(* CODESYS project RobotArm.project

Project tree, tasks and I/O mapping:
  Device : CODESYS Control for Raspberry Pi SL, 3S - Smart Software Solutions GmbH, version 3.5.12.0
    application Application
      libraries: Standard, * (System); SysProcess, 3.5.7.0 (System); SysTypes Interfaces, 3.5.2.0 (System)
      task MainTask (cyclic, interval t#10ms, priority 1) calls PLC_PRG
      task VISU_TASK (cyclic, interval 100 ms, priority 31) calls VisuElems.Visu_Prg
      program PLC_PRG [ST]
      program prgModeSelect [ST]
      program prgStartup [CFC]
      visualisation Visualization
      GVLs/
        global variables GVL_IO
        global variables GVL_Constants
        global variables GVL_Axis
      DUTs/
        data type eAxis
      FBs/
        function block fb_AxisControl [CFC]
        function block fb_FreeMode [SFC]: MoveA_active, MoveA_exit, Check_active
      program prgAxisControl [ST]
    SoftMotion General Axis Pool
    I²C
      I2C_master : I2C master, 3S - Smart Software Solutions GmbH, version 1.0.0.0
        Adafruit_PWM_SoftMotion : Adafruit PWM SoftMotion, 3S - Smart Software Solutions GmbH, version 1.2.0.0
            settings: I²C address = 16#40; Frequency [Hz] = 60
          SM_Drive_Servo_Base : SM_Drive_Servo, 3S - Smart Software Solutions GmbH, version 3.5.11.0
              settings: wDriveID = 0; fSWMaxVelocity = 1000; Commisioning.smci.Distance = 10; Commisioning.smci.Velocity = 30; Commisioning.smci.Acceleration = 500; Commisioning.smci.Deceleration = 500; negative position [units] = -90; positive position [units] = 100; minimum signal length [ms] = 0.5; maximum signal length [ms] representing the positive position = 2.2
          SM_Drive_Servo_Upright : SM_Drive_Servo, 3S - Smart Software Solutions GmbH, version 3.5.11.0
              settings: fSWMaxVelocity = 1000; negative position [units] = -90; positive position [units] = 100; minimum signal length [ms] = 0.5; maximum signal length [ms] representing the positive position = 2.2
          SM_Drive_Servo_Arm : SM_Drive_Servo, 3S - Smart Software Solutions GmbH, version 3.5.11.0
              settings: wDriveID = 2; fSWMaxVelocity = 1000
          SM_Drive_Servo_Gripper : SM_Drive_Servo, 3S - Smart Software Solutions GmbH, version 3.5.11.0
              settings: wDriveID = 3; fSWMaxVelocity = 1000
    SPI
    GPIOs_A_B : GPIOs B+/Pi2, 3S - Smart Software Solutions GmbH, version 3.5.11.0
        unmapped channels: digital inputs (GPIO0..GPIO31), digital outputs (GPIO0..GPIO31)
    Onewire
    Camera device
      <Empty>
  text list GlobalTextList
*)

// Device/Application/DUTs/eAxis
TYPE eAxis :
(
	Base := 1,
	Upright := 2,
	Arm := 3,
	Gripper := 4
);
END_TYPE

// Device/Application/GVLs/GVL_IO
VAR_GLOBAL
	rVelocity : LREAL := 100;
	rPos : ARRAY [1..iNoOfAxis] OF LREAL;
END_VAR

// Device/Application/GVLs/GVL_Constants
VAR_GLOBAL CONSTANT
	iNoOfAxis: INT := 4;
END_VAR

// Device/Application/GVLs/GVL_Axis
VAR_GLOBAL
	fbAxisControl: ARRAY [1..iNoOfAxis] OF fb_AxisControl;
END_VAR

// Device/Application/PLC_PRG
PROGRAM PLC_PRG
VAR_INPUT
	bStartup: BOOL;
END_VAR
VAR
	bShutdown: BOOL;
	stdout : STRING(1000) := '';	
	Result : RTS_IEC_RESULT;
END_VAR

IF NOT bStartup THEN
	prgStartup();
END_IF

IF bStartup THEN
	prgAxisControl();
	prgModeSelect();
END_IF

IF bShutdown THEN
	bShutdown := FALSE;
	SysProcess.SysProcessExecuteCommand2(pszCommand:='sudo shutdown -h now', pszStdOut:=stdout, udiStdOutLen:= SIZEOF(stdout),pResult := ADR(Result));
END_IF

END_PROGRAM

// Device/Application/prgStartup
PROGRAM prgStartup
VAR
	MC_Power_Base: MC_Power;
	MC_Power_Upright: MC_Power;
	MC_Power_Arm: MC_Power;
	MC_Power_Gripper: MC_Power;
END_VAR

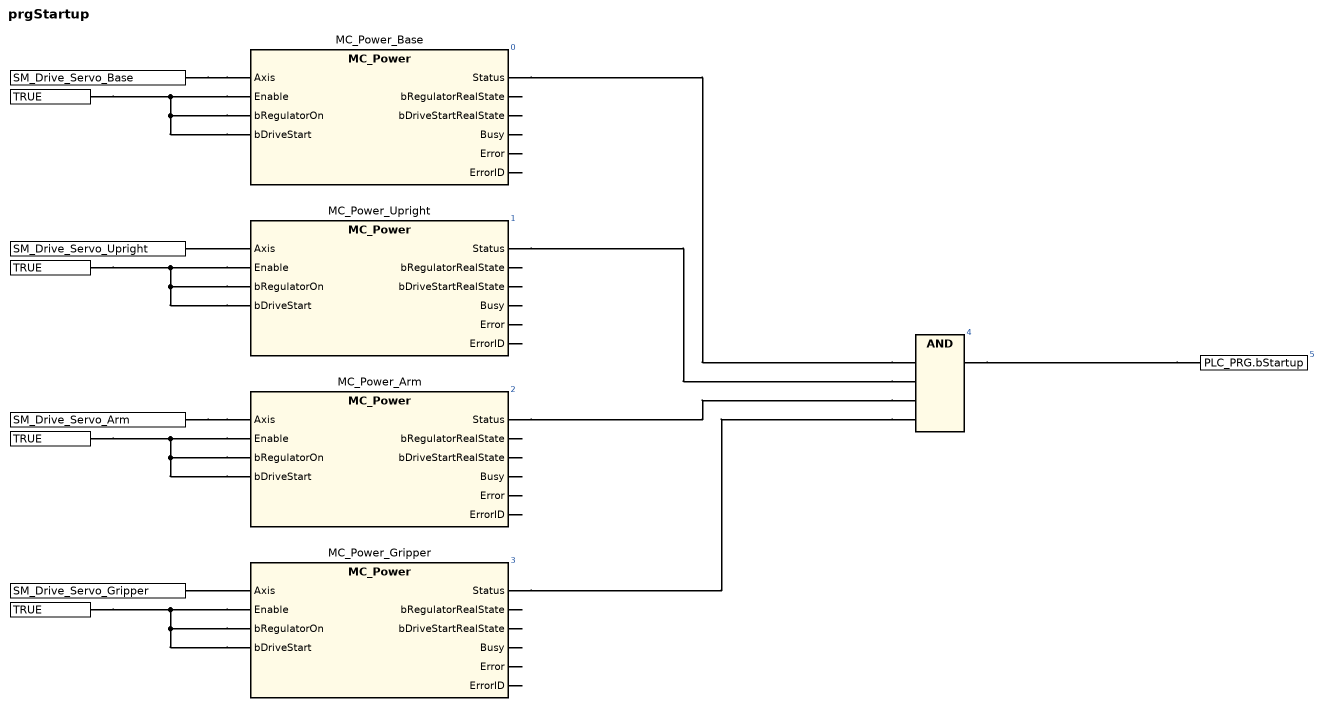
// note: 5 stored wires end on pins the file does not list and are not shown
MC_Power_Base(Axis := SM_Drive_Servo_Base, Enable := TRUE, bRegulatorOn := TRUE, bDriveStart := TRUE); // MC_Power
MC_Power_Upright(Axis := SM_Drive_Servo_Upright, Enable := TRUE, bRegulatorOn := TRUE, bDriveStart := TRUE); // MC_Power
MC_Power_Arm(Axis := SM_Drive_Servo_Arm, Enable := TRUE, bRegulatorOn := TRUE, bDriveStart := TRUE); // MC_Power
MC_Power_Gripper(Axis := SM_Drive_Servo_Gripper, Enable := TRUE, bRegulatorOn := TRUE, bDriveStart := TRUE); // MC_Power
PLC_PRG.bStartup := MC_Power_Base.Status AND MC_Power_Upright.Status AND MC_Power_Arm.Status AND MC_Power_Gripper.Status;

END_PROGRAM

// Device/Application/prgAxisControl
PROGRAM prgAxisControl
VAR
END_VAR

fbAxisControl[Base](Axis:=SM_Drive_Servo_Base);
fbAxisControl[Upright](Axis:=SM_Drive_Servo_Upright);
fbAxisControl[Arm](Axis:=SM_Drive_Servo_Arm);
fbAxisControl[Gripper](Axis:=SM_Drive_Servo_Gripper);

END_PROGRAM

// Device/Application/prgModeSelect
PROGRAM prgModeSelect
VAR
	Axis : INT;
	fbFreeMode: ARRAY [1..iNoOfAxis] of fb_FreeMode;
END_VAR

//Free Mode
FOR Axis := 1 TO iNoOfAxis DO
	fbFreeMode[Axis](Axis := Axis, rPos := rPos[Axis]);
END_FOR

END_PROGRAM

// Device/Application/FBs/fb_FreeMode
FUNCTION_BLOCK fb_FreeMode
VAR_INPUT
	rPos: LREAL;
	Axis :INT;
END_VAR
VAR_OUTPUT
END_VAR
VAR
	bNewPos: BOOL;
END_VAR

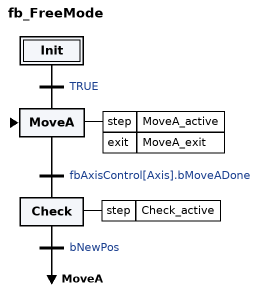
INITIAL_STEP Init:
END_STEP
TRANSITION FROM Init TO MoveA
    := TRUE;
END_TRANSITION
STEP MoveA:
    MoveA_active(N);  // step action
    MoveA_exit(P0);  // exit action
END_STEP
TRANSITION FROM MoveA TO Check
    := fbAxisControl[Axis].bMoveADone;
END_TRANSITION
STEP Check:
    Check_active(N);  // step action
END_STEP
TRANSITION FROM Check TO MoveA
    := bNewPos;
END_TRANSITION

ACTION MoveA_active:
fbAxisControl[Axis].rMoveAPos := rPos;
fbAxisControl[Axis].rMoveAVel := rVelocity;
fbAxisControl[Axis].rMoveAAcc := 500;
fbAxisControl[Axis].rMoveADec := 500;
fbAxisControl[Axis].bMoveA := TRUE;
END_ACTION

ACTION MoveA_exit:
fbAxisControl[Axis].bMoveA := FALSE;
END_ACTION

ACTION Check_active:
IF rPos <> fbAxisControl[Axis].rActualPos THEN
	bNewPos := TRUE;
ELSE
	bNewPos := FALSE;
END_IF
END_ACTION

END_FUNCTION_BLOCK

// Device/Application/FBs/fb_AxisControl
FUNCTION_BLOCK fb_AxisControl
VAR_INPUT
	bMoveA: BOOL;
	rMoveAPos: LREAL;
	rMoveAVel: LREAL;
	rMoveAAcc: LREAL;
	rMoveADec: LREAL;
END_VAR
VAR_OUTPUT
	bMoveADone: BOOL;				(*Axis Absolute Move is complete*)
	bMoveABusy: BOOL;				(*Axis Absolute Move is Busy*)
	bMoveAAborted: BOOL;				(*Axis Absolute Move was Aborted*)
	bMoveAError: BOOL;				(*Axis Absolute Move error occurred*)
	eIDMoveAError: UDINT;			(*Error ID for the Axis Absolute Move Error*)
	rActualPos: LREAL;
END_VAR
VAR
	mcMoveAbs: MC_MoveAbsolute;
END_VAR
VAR_IN_OUT
	Axis : AXIS_REF_SERVO;
END_VAR

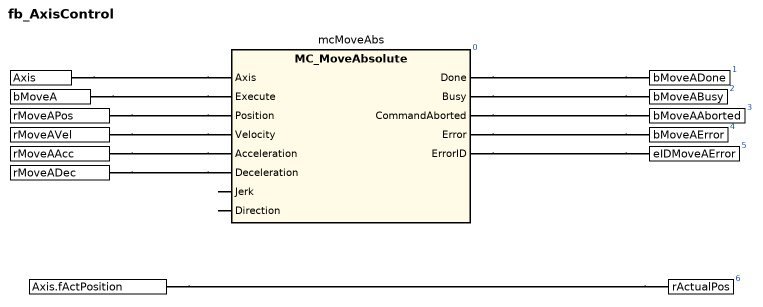
mcMoveAbs(
    Axis := Axis,
    Execute := bMoveA,
    Position := rMoveAPos,
    Velocity := rMoveAVel,
    Acceleration := rMoveAAcc,
    Deceleration := rMoveADec); // MC_MoveAbsolute
bMoveADone := mcMoveAbs.Done;
bMoveABusy := mcMoveAbs.Busy;
bMoveAAborted := mcMoveAbs.CommandAborted;
bMoveAError := mcMoveAbs.Error;
eIDMoveAError := mcMoveAbs.ErrorID;
rActualPos := Axis.fActPosition;

END_FUNCTION_BLOCK

// Device/Application/Visualization
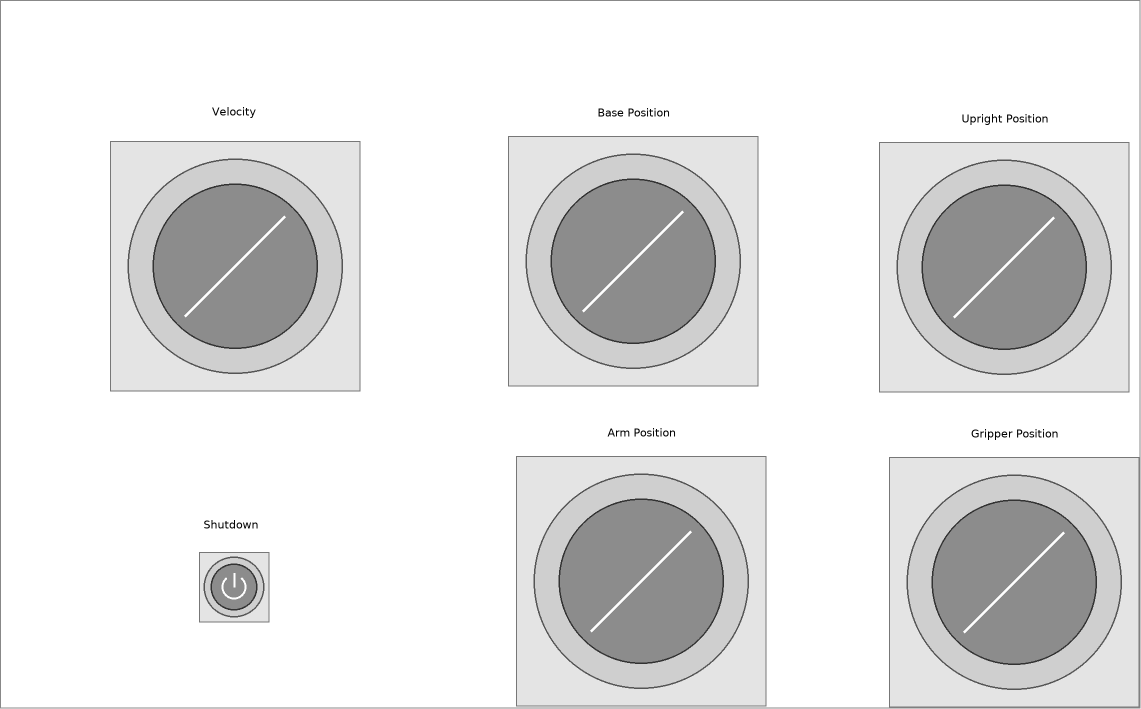
VISUALIZATION Visualization  // 1141x709
    Potentiometer360 (110,141 250x250), variable: rVelocity, style: Potentiometer-Potentiometer360-Gray, scale format: %.1f, scale 10..510
        p2431819421: Outside
    Label (159,97 150x30), "Velocity"
    Label (559,98 150x30), "Base Position"
    Potentiometer360 (508,136 250x250), variable: rPos[Base], style: Potentiometer-Potentiometer360-Gray, scale format: %.1f, scale -90..90
        p2431819421: Outside
    Label (930,104 150x30), "Upright Position"
    Potentiometer360 (879,142 250x250), variable: rPos[Upright], style: Potentiometer-Potentiometer360-Gray, scale format: %.1f, scale -40..60
        p2431819421: Outside
    Label (567,418 150x30), "Arm Position"
    Potentiometer360 (516,456 250x250), variable: rPos[Arm], style: Potentiometer-Potentiometer360-Gray, scale format: %.1f, scale -60..60
        p2431819421: Outside
    Label (940,419 150x30), "Gripper Position"
    Potentiometer360 (889,457 250x250), variable: rPos[Gripper], style: Potentiometer-Potentiometer360-Gray, scale format: %.1f, scale -60..60
        p2431819421: Outside
    PowerSwitch (199,552 70x70), variable: PLC_PRG.bShutdown, behaviour: TOGGLE, style: Switch-PowerSwitch-Gray
    Label (156,510 150x30), "Shutdown"
END_VISUALIZATION
